# EPICS substitutions: mc07/tpmacApp/pmc/xf16idc-mc07-homing.substitutions
file "home_to_enc_ref_template.pmc"
{

pattern
{ AXIS,   PLC,  SERVO,  TIMER }
#{ 1,      8,    701,    5511  }
#{ 2,      9,    702,    5512  }
#{ 3,      10,   703,    5611  }
#{ 4,      11,   704,    5612  }
#{ 5,      12,   711,    5711  }
#{ 6,      13,   712,    5712  }
#{ 7,      14,   713,    5811  }
#{8,	15,	714,	5812}
}

file "home_to_limit_template.pmc"
{
pattern
{ AXIS,   PLC,  SERVO,  TIMER }
{ 1,      8,    701,    5511  }
{ 2,      9,    702,    5512  }
{ 3,      10,   703,    5611  }
{ 4,      11,   704,    5612  }
#{ 6,      13,   712,    5712  }
#{ 7,      14,   713,    5811  }
}
